TYPE CyclicAxis_Param_typ :
STRUCT
	
	ThreadName		: STRING[20];
	CyclicPos		: CyclicPos_Param_typ;
    CyclicVel		: CyclicVel_Param_typ;   
END_STRUCT
END_TYPE

(* stored: Version 1.1.0.1, ProductVersion 3.1.4024.3
   DUT CyclicAxis_Param_typ: Id {a28676e0-5f96-021b-10e3-a80229e8d70e} *)
